PROGRAM MAIN
VAR
	diKapasativSensor1 AT %I* : BOOL ;
	bMinneKapasativSensor1 : BOOL := 0 ;
	diKapasativSensor2 AT %I* : BOOL ;
	bMinneKapasativSensor2 : BOOL := 0 ;
	AndMinne : BOOL := 0 ;
	OrMinne : BOOL := 0 ;
END_VAR

bMinneKapasativSensor1 := diKapasativSensor1 ;
bMinneKapasativSensor2 := diKapasativSensor2 ;
AndMinne := diKapasativSensor1 AND diKapasativSensor2 ;
OrMinne := diKapasativSensor1 XOR diKapasativSensor2 ;

END_PROGRAM

(* stored: Version 1.1.0.1, ProductVersion 3.1.4024.9
   POU MAIN: Id {72cf5da1-53fe-433c-ac52-4d53f2dfe827}, SpecialFunc None *)
